(* IEC 61131-3 sources: test/Class/HmiAsciiBuffer, 1 file *)

(* ---- HmiAsciiBuffer.st ---- *)
(*!
<Class
	Name               = "HmiAsciiBuffer"
	Revision           = "0.1"
	RealtimeTask       = "false"
	CyclicTask         = "false"
	BackgroundTask     = "false"
	Sigmatek           = "true"
	OSInterface        = "false"
	HighPriority       = "false"
	Automatic          = "false"
	UpdateMode         = "Prescan"
	SharedCommandTable = "true"
	Objectsize         = "(284,120)">
	<Channels>
		<Server Name="ClassSvr" Visualized="false" Initialize="false" WriteProtected="true" Retentive="false"/>
		<Client Name="File" Required="true" Internal="false"/>
		<Client Name="StringLib" Required="true" Internal="false"/>
	</Channels>
	<RevDoku>
		<Owner Company="sigmatek" Author="kolott"/>
		<Dokumentation Revision="0.1" Date="2018-12-27" Author="kolott" Company="sigmatek" Description="Method RenText() added"/>
	</RevDoku>
</Class>
*)
HmiAsciiBuffer : CLASS
  //Servers:
	ClassSvr 	: SvrChCmd_DINT;
  //Clients:
	File 	: CltChCmd_HmiFile;
	StringLib 	: CltChCmd_HmiStrLib;
  //Variables:
		Default 	: CHAR;
		No 	: UDINT;
		Ptr 	: ^CHAR;
		Change 	: BOOL;
		Size 	: UDINT;
		GuidePost 	: ^UDINT;
  //Functions:

	FUNCTION HmiAsciiBuffer
		VAR_OUTPUT
			ret_code 	: ConfStates;
		END_VAR;

	FUNCTION GLOBAL GetText
		VAR_INPUT
			txtno 	: UDINT;
		END_VAR
		VAR_OUTPUT
			retcode 	: ^CHAR;
		END_VAR;

	FUNCTION GLOBAL AddText
		VAR_INPUT
			src 	: ^CHAR;
		END_VAR
		VAR_OUTPUT
			retcode 	: BOOL;
		END_VAR;

	FUNCTION GLOBAL Free;

	FUNCTION GLOBAL Load
		VAR_OUTPUT
			retcode 	: BOOL;
		END_VAR;

	FUNCTION GLOBAL GetNo
		VAR_OUTPUT
			retcode 	: UDINT;
		END_VAR;

	FUNCTION GLOBAL MakeGuidePost;

	FUNCTION GLOBAL KillGuidePost;

	FUNCTION GLOBAL GetNoByName
		VAR_INPUT
			name 	: ^CHAR;
		END_VAR
		VAR_OUTPUT
			retcode 	: UDINT;
		END_VAR;

	FUNCTION GLOBAL OverloadLight
		VAR_INPUT
			xxno 	: DINT;
		END_VAR;

	FUNCTION GLOBAL RenText
		VAR_INPUT
			txtno 	: UDINT;
			psrc 	: ^CHAR;
		END_VAR
		VAR_OUTPUT
			retcode 	: BOOL;
		END_VAR;
  //Tables:
	FUNCTION @STD
		VAR_OUTPUT
			ret_code	: CONFSTATES;
		END_VAR;
	FUNCTION GLOBAL TAB @CT_;
END_CLASS;

#pragma usingLtd HmiFile
#pragma usingLtd HmiStrLib

FUNCTION HmiAsciiBuffer::HmiAsciiBuffer
	VAR_OUTPUT
		ret_code 	: ConfStates;
	END_VAR

	ret_code := C_OK;

  Ptr := NIL;
  No := 0;
  Default := 0;
  Change := false;
  Size := 0;
  GuidePost := NIL;

END_FUNCTION

FUNCTION GLOBAL HmiAsciiBuffer::GetText
	VAR_INPUT
		txtno 	: UDINT;
	END_VAR
	VAR_OUTPUT
		retcode 	: ^char;
	END_VAR
  var
    ph : ^udint;
  end_var

  retcode := #Default;

  if(Ptr <> NIL) then
    if(txtno < No) then
      if(GuidePost = NIL) then
        retcode := Ptr;
        while(txtno) do
          txtno   -= 1;
          retcode += (StringLib.StrLen(retcode, sizeof(char)) + sizeof(char));
        end_while;
      else
        ph      := GuidePost + (4 * txtno);
        retcode := Ptr + ph^;
      end_if;
    end_if;
  end_if;

END_FUNCTION

FUNCTION GLOBAL HmiAsciiBuffer::AddText
	VAR_INPUT
		src 	: ^char;
	END_VAR
	VAR_OUTPUT
		retcode 	: BOOL;
	END_VAR
  var
    len : udint;
    tmp : udint;
  end_var;

  retcode := false;
  len     := StringLib.StrLen(src, sizeof(char)) + 1;
  tmp     := Size + len;

  if(StringLib.XMemory(#Ptr, tmp) = true) then
 	  StringLib.StrCpy(Ptr + Size, sizeof(char), src, sizeof(char));
	  No      += 1;
	  Size    := tmp;
	  Change  := true;
    retcode := true;
    KillGuidePost();
  end_if;

END_FUNCTION

FUNCTION GLOBAL HmiAsciiBuffer::Free

  KillGuidePost();
  StringLib.XMemory(#Ptr, 0);
  Ptr := NIL;
  No := 0;
  Default := 0;
  Change := false;
  Size := 0;
  ClassSvr := 0;

END_FUNCTION

FUNCTION GLOBAL HmiAsciiBuffer::Load
	VAR_OUTPUT
		retcode 	: BOOL;
	END_VAR
  var
    chrsize : usint;
    txtno : udint;
    txtsize : udint;
  end_var

	// [] .......... sizeof character
	// [][][][] .... no of text (ab compiler version 32 4byte, vorher 2byte)
	// [][][][] .... no of characters
	// [ ........... text

  retcode := false;
  Free();

  File.FRead(#chrsize, 1);
  File.FRead(#txtno, 4);
  File.FRead(#txtsize, 4);

  if(File.FChkFile() = true) then
    if(chrsize = sizeof(char)) then
      File.FMemory(#Ptr, txtsize);
      File.FRead(Ptr, txtsize);

      if(File.FChkFile() = true) then
        Size    := txtsize;
        No      := txtno;
        retcode := true;
      else
        Free();
      end_if;
    end_if;
  end_if;

  ClassSvr := to_dint(No);

END_FUNCTION

FUNCTION GLOBAL HmiAsciiBuffer::GetNo
	VAR_OUTPUT
		retcode 	: UDINT;
	END_VAR

  retcode := No;

END_FUNCTION

FUNCTION GLOBAL HmiAsciiBuffer::MakeGuidePost

  StringLib.MakeGuidePost(#GuidePost, Ptr, No, sizeof(char));

END_FUNCTION

FUNCTION GLOBAL HmiAsciiBuffer::KillGuidePost

  StringLib.XMemory(#GuidePost, 0);

END_FUNCTION

FUNCTION GLOBAL HmiAsciiBuffer::GetNoByName
	VAR_INPUT
		name 	: ^char;
	END_VAR
	VAR_OUTPUT
		retcode 	: UDINT;
	END_VAR
  var
    chr : char;
    ph : ^char;
    poff : ^udint;
    txtno : udint;
  end_var

  if(Ptr <> NIL)&(No > 0) then
    txtno := No;
    chr   := name^;

    if(GuidePost = NIL) then
      ph := Ptr;
      while(txtno) do
        if(ph^ = chr) then
          if(StringLib.StrCmp(ph, sizeof(char), name, sizeof(char)) = 0) then
            retcode := No - txtno;
            return;
          end_if;
        end_if;
        ph += (StringLib.StrLen(ph, sizeof(char)) + sizeof(char));
        txtno -= 1;
      end_while;
    else
      retcode := 0;
      poff    := GuidePost;
      while(txtno) do
        ph := Ptr + poff^;
        if(ph^ = chr) then
          if(StringLib.StrCmp(ph, sizeof(char), name, sizeof(char)) = 0) then
            return;
          end_if;
        end_if;
        retcode += 1;
        txtno   -= 1;
        poff    += 4;
      end_while;
    end_if;
  end_if;

  retcode := 16#FFFFFFFF;

END_FUNCTION

FUNCTION GLOBAL HmiAsciiBuffer::OverloadLight
	VAR_INPUT
		xxno 	: DINT;
	END_VAR
  var
    ph : ^usint;
    anz : udint;
  end_var

  if(Size > 1) then

    ph  := Ptr;
    anz := Size - 1;

    while(anz) do
      if(ph$^uint^ = 0x5858) then
        ph^ := '0' + (xxno$usint / 10);
        ph  += 1;
        ph^ := '0' + (xxno$usint mod 10);
      end_if;
      ph  += 1;
      anz -= 1;
    end_while;
  end_if;

END_FUNCTION

FUNCTION GLOBAL HmiAsciiBuffer::RenText
	VAR_INPUT
    txtno : udint;
		psrc 	: ^char;
	END_VAR
	VAR_OUTPUT
		retcode 	: BOOL;
	END_VAR
  var
    ptxt : ^char;
    len0, len1 : udint;
    offset, rest : udint;
  end_var;

  retcode := false;
  ptxt    := GetText(txtno);

  if((ptxt <> NIL) & (psrc <> NIL)) then
    len0 := StringLib.StrLen(ptxt, sizeof(char)) + 1;
    len1 := StringLib.StrLen(psrc, sizeof(char)) + 1;

    if(len0 = len1) then // keep size
      if(StringLib.StrCmp(ptxt, sizeof(char), psrc, sizeof(char)) <> 0) then
        StringLib.StrCpy(ptxt, sizeof(char), psrc, sizeof(char));
        Change := true;
      end_if;
      retcode := true;
    elsif(len0 > len1) then // downsize
      StringLib.StrCpy(ptxt, sizeof(char), psrc, sizeof(char));
      offset := ptxt$udint - Ptr$udint;
      rest   := Size - offset - len0;
      _memmove(ptxt+len1, ptxt+len0, rest);
      Size   := Size + len1 - len0;
      if(GuidePost <> NIL) then
        MakeGuidePost();
      end_if;
      Change  := true;
      retcode := true;
    else // upsize
      offset := ptxt$udint - Ptr$udint;
      if(StringLib.XMemory(#Ptr, Size - len0 + len1) = true) then
        ptxt   := Ptr + offset; // correct ptxt
        rest   := Size - offset - len0;
        _memmove(Ptr+offset+len1, Ptr+offset+len0, rest);
        StringLib.StrCpy(ptxt, sizeof(char), psrc, sizeof(char));
        Size := Size + len1 - len0;
        if(GuidePost <> NIL) then
          MakeGuidePost();
        end_if;
        Change  := true;
        retcode := true;
      end_if;
    end_if;
  end_if;

END_FUNCTION
